// TIA Portal V20 export
DATA_BLOCK "DB_ConveyorParameters"   // DB6
// stored: Access Published, MemoryReserve 100, Namespace ProductionLine
   VAR
      ProductionLine : Struct
         Conveyor : Array[_.minProductionLine.._.maxProductionLine] of "Global.ConveyorParameters";
         MABS { S7_SetPoint := 'True'} : Array[_."A1.9.1".._."A1.6.2"] of "Global.MABS_Parameters";
         TransferUnit { S7_SetPoint := 'True'} : Array[_."A1.13.1".._."D1.10.1"] of "Global.ConveyorParameters_TransferUnit";
      END_STRUCT;
   END_VAR
BEGIN
END_DATA_BLOCK
